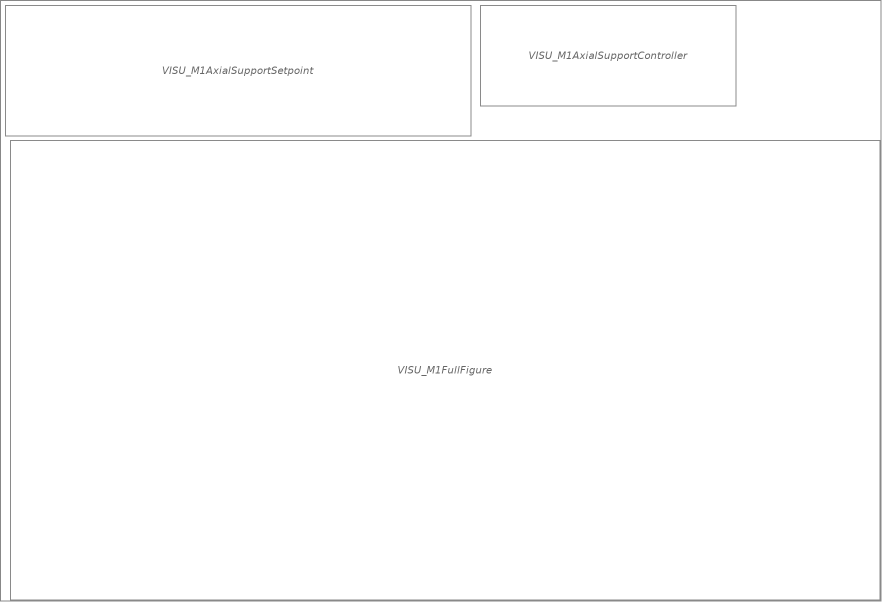
VISUALIZATION VISU_M1AxialSupport  // 882x602
VAR_IN_OUT
	ref : M1AxialSupport;
    widget : M1AxialSupportWidget;
    m1Ref : M1;
    m1Widget : M1Widget;
END_VAR
    Frame (5,5 466x131)
        shows VISU_M1AxialSupportSetpoint(ref := ref, widget := widget)
    Frame (10,140 870x460)
        shows VISU_M1FullFigure(ref := m1Ref, widget := m1Widget)
    Frame (480,5 256x101)
        shows VISU_M1AxialSupportController(ref := ref, widget := widget)
END_VISUALIZATION

(* stored: Version 1.1.0.1, ProductVersion 3.1.4019.2
   Visu VISU_M1AxialSupport: Id {3d3d77fe-480b-4328-90fa-41e5a4aecea9} *)
